PROGRAM Rotina021_Manual
VAR
	status: INT;
	
	posicaoAtual: STRING;
	envialog: STRING;
	
	fbTimeVentila: ton;
	fbTimeAqueci: ton;
	
	totalManual: STRING(255);
	tempo: STRING(255);
	
	Estufa: INT;
	
END_VAR

fbTimeVentila();
fbTimeAqueci();
Estufa:= 2;

CASE status OF

0:
IF gvl_p.arrStatusEstufas[Estufa].startManual AND STRING_TO_DT(gvl.progInicio[Estufa]) <= systemtime_to_dt(gvl.fbGetLocalSystemTime.systemTime)  THEN
	status:= 5;
	
	gvl.bstartchart021:= TRUE;
	gvl_p.zona1setpt_021:= gvl_p.arr_CustomTime_021[0,1];
	gvl_p.zona2setpt_021:= gvl_p.arr_CustomTime_021[0,1];
	gvl.liga_ventilacao_021:= TRUE;
	fbTimeVentila(in:= TRUE, pt:=T#1S);
	
///// GERADOR DE LOG -------------------------------------------------------------

envialog:= 'Programação Manual Iniciada ESTUFA 021';
gvl.logRegister21:= envialog;
	
	gvl_p.etapa_process[Estufa] := 'Inicializando';
	
ELSE
	status:= 0;
	IF gvl_p.arrStatusEstufas[Estufa].start THEN
		gvl_p.etapa_process[Estufa] := gvl.progInicio[Estufa];
	END_IF
END_IF
5:
IF fbTimeVentila.Q THEN
	status:= 10;
	gvl.liga_ventilacao_021:=FALSE;
	fbTimeVentila(in:= FALSE);
ELSE
	status:= 5;
END_IF

10:
IF gvl.ventilacao_Ligada_021 THEN
	status:= 15;
	
	gvl.liga_aquecimento_021:= TRUE;
	fbTimeAqueci(in:= TRUE, pt:= T#1S);
	
///// GERADOR DE LOG -------------------------------------------------------------

envialog:= 'Aquecendo ESTUFA 021';
gvl.logRegister21:= envialog;

	gvl_p.etapa_process[Estufa] := 'Aquecendo';
	
ELSE
	status:= 10;
END_IF

15:
IF fbTimeAqueci.Q THEN
	status:= 20;
	
	gvl.liga_aquecimento_021:= FALSE;
	fbTimeAqueci(in:=false);
ELSE
	status:= 15;
END_IF

20:
IF gvl.zona1atual_021 >= gvl_p.zona1setpt_021 THEN
	status:= 30;
	
gvl.progInicio[Estufa]:= DT_TO_STRING(gvl.somaTempo);
	
///// CALCULAR FIM DA SECAGEM E DA ARMAZENAGEM --------------------------------------------------------------------------------

totalManual:= insert('T#h',INT_TO_STRING(gvl.totalManual[Estufa]),2);
gvl_p.arrStatusEstufas[Estufa].inicioSecagem := STRING_TO_DT(gvl.progInicio[Estufa]);
gvl_p.arrStatusEstufas[Estufa].fimSecagem := STRING_TO_DT(gvl.progInicio[Estufa]) + STRING_TO_TIME(totalManual);
gvl_P.arrStatusEstufas[Estufa].prevFimSeca := gvl_p.arrStatusEstufas[Estufa].fimSecagem;
//gvl_p.arrStatusEstufas[0].fimArmazenagem := gvl_p.arrStatusEstufas[0].fimSecagem + gvl_p.arrStatusEstufas[0].tempoArmazenagem ;

///// IMPRIMIR A HORA E A DATA DO INICIO DA SECAGEM ---------------------------------------------------------------------------
gvl_p.arrStatusEstufas[Estufa].statusInicioSecagem := '';
gvl_p.arrStatusEstufas[Estufa].statusInicioSecagem := concat(gvl_p.arrStatusEstufas[Estufa].statusInicioSecagem,gvl.hora);
gvl_p.arrStatusEstufas[Estufa].statusInicioSecagem := concat(gvl_p.arrStatusEstufas[Estufa].statusInicioSecagem,':');
gvl_p.arrStatusEstufas[Estufa].statusInicioSecagem := concat(gvl_p.arrStatusEstufas[Estufa].statusInicioSecagem,gvl.minuto);
gvl_p.arrStatusEstufas[Estufa].statusInicioSecagem := concat(gvl_p.arrStatusEstufas[Estufa].statusInicioSecagem,' ');
gvl_p.arrStatusEstufas[Estufa].statusInicioSecagem := concat(gvl_p.arrStatusEstufas[Estufa].statusInicioSecagem,gvl.dia);
gvl_p.arrStatusEstufas[Estufa].statusInicioSecagem := concat(gvl_p.arrStatusEstufas[Estufa].statusInicioSecagem,'/');
gvl_p.arrStatusEstufas[Estufa].statusInicioSecagem := concat(gvl_p.arrStatusEstufas[Estufa].statusInicioSecagem,gvl.mes);
gvl_p.arrStatusEstufas[Estufa].statusInicioSecagem := concat(gvl_p.arrStatusEstufas[Estufa].statusInicioSecagem,'/');
gvl_p.arrStatusEstufas[Estufa].statusInicioSecagem := concat(gvl_p.arrStatusEstufas[Estufa].statusInicioSecagem,gvl.ano);

//--------------------REATOR------------------------------------

IF gravarConfigPosicao_Reator.bGravarConfigPosicao_Reator THEN
	gvl_p.arrStatusEstufas[Estufa].inicioReator := '';
	gvl_p.arrStatusEstufas[Estufa].inicioReator := concat(gvl_p.arrStatusEstufas[Estufa].inicioReator,gvl.hora);
	gvl_p.arrStatusEstufas[Estufa].inicioReator := concat(gvl_p.arrStatusEstufas[Estufa].inicioReator,':');
	gvl_p.arrStatusEstufas[Estufa].inicioReator := concat(gvl_p.arrStatusEstufas[Estufa].inicioReator,gvl.minuto);
	gvl_p.arrStatusEstufas[Estufa].inicioReator := concat(gvl_p.arrStatusEstufas[Estufa].inicioReator,' ');
	gvl_p.arrStatusEstufas[Estufa].inicioReator := concat(gvl_p.arrStatusEstufas[Estufa].inicioReator,gvl.dia);
	gvl_p.arrStatusEstufas[Estufa].inicioReator := concat(gvl_p.arrStatusEstufas[Estufa].inicioReator,'/');
	gvl_p.arrStatusEstufas[Estufa].inicioReator := concat(gvl_p.arrStatusEstufas[Estufa].inicioReator,gvl.mes);
	gvl_p.arrStatusEstufas[Estufa].inicioReator := concat(gvl_p.arrStatusEstufas[Estufa].inicioReator,'/');
	gvl_P.arrStatusEstufas[Estufa].inicioReator := concat(gvl_p.arrStatusEstufas[Estufa].inicioReator,gvl.ano);
END_IF

///// DECOMPOR A VARIAVEL FIM DA SECAGEM -----------------------------------------------------------------------------------------------
gvl_p.arrStatusEstufas[Estufa].diaSec := MID(STR:= DT_TO_STRING(gvl_p.arrStatusEstufas[Estufa].fimSecagem) , LEN:= 2, POS:=12);
gvl_p.arrStatusEstufas[Estufa].mesSec := MID(STR:= DT_TO_STRING(gvl_p.arrStatusEstufas[Estufa].fimSecagem), LEN:= 2, POS:=9);
gvl_p.arrStatusEstufas[Estufa].anoSec := MID(STR:= DT_TO_STRING(gvl_p.arrStatusEstufas[Estufa].fimSecagem), LEN:= 2, POS:=6);
gvl_p.arrStatusEstufas[Estufa].horaSec := MID(STR:= DT_TO_STRING(gvl_p.arrStatusEstufas[Estufa].fimSecagem), LEN:= 2, POS:=15);
gvl_p.arrStatusEstufas[Estufa].minutoSec := MID(STR:= DT_TO_STRING(gvl_p.arrStatusEstufas[Estufa].fimSecagem), LEN:= 2, POS:=18);

///// IMPRIMIR A HORA E A DATA DO FIM DA SECAGEM --------------------------------------------------------------------------------------------------------
gvl_p.arrStatusEstufas[Estufa].statusFimSecagem := '';
gvl_p.arrStatusEstufas[Estufa].statusFimSecagem := concat(gvl_p.arrStatusEstufas[Estufa].statusFimSecagem,gvl_p.arrStatusEstufas[0].horaSec);
gvl_p.arrStatusEstufas[Estufa].statusFimSecagem := concat(gvl_p.arrStatusEstufas[Estufa].statusFimSecagem,':');
gvl_p.arrStatusEstufas[Estufa].statusFimSecagem := concat(gvl_p.arrStatusEstufas[Estufa].statusFimSecagem,gvl_p.arrStatusEstufas[0].minutoSec);
gvl_p.arrStatusEstufas[Estufa].statusFimSecagem := concat(gvl_p.arrStatusEstufas[Estufa].statusFimSecagem,' ');
gvl_p.arrStatusEstufas[Estufa].statusFimSecagem := concat(gvl_p.arrStatusEstufas[Estufa].statusFimSecagem,gvl_p.arrStatusEstufas[0].diaSec);
gvl_p.arrStatusEstufas[Estufa].statusFimSecagem := concat(gvl_p.arrStatusEstufas[Estufa].statusFimSecagem,'/');
gvl_p.arrStatusEstufas[Estufa].statusFimSecagem := concat(gvl_p.arrStatusEstufas[Estufa].statusFimSecagem,gvl_p.arrStatusEstufas[0].mesSec);
gvl_p.arrStatusEstufas[Estufa].statusFimSecagem := concat(gvl_p.arrStatusEstufas[Estufa].statusFimSecagem,'/');
gvl_p.arrStatusEstufas[Estufa].statusFimSecagem := concat(gvl_p.arrStatusEstufas[Estufa].statusFimSecagem,gvl_p.arrStatusEstufas[0].anoSec);


///// GERADOR DE LOG -------------------------------------------------------------
envialog:= 'Inicio T1 ESTUFA 021';
gvl.logRegister21:= envialog;

gvl_p.etapa_process[2]:= 'T1';

ELSE
	IF gvl_p.arr_CustomTime_021[1,1] = 0 THEN
		status:= 45;
	END_IF
	status:= 20;
END_IF

30:
tempo:= insert('T#h',INT_TO_STRING(gvl_p.arr_CustomTime_021[1,1]),2);
IF STRING_TO_DT(gvl.progInicio[Estufa]) + STRING_TO_TIME(tempo) = systemtime_to_dt(gvl.fbGetLocalSystemTime.systemTime) THEN
	status:= 31;
	
	gvl_p.zona1setpt_021:= gvl_p.arr_CustomTime_021[0,2];
	gvl_p.zona2setpt_021:= gvl_p.arr_CustomTime_021[0,2];
	gvl.progInicio[Estufa]:= DT_TO_STRING(STRING_TO_DT(gvl.progInicio[Estufa]) + STRING_TO_TIME(tempo));
	
///// GERADOR DE LOG -------------------------------------------------------------
envialog:= 'Inicio T2 ESTUFA 021';
gvl.logRegister21:= envialog;

gvl_p.etapa_process[2]:= 'T2';
	
ELSE
	status:= 30;
END_IF

31:
tempo:= insert('T#h',INT_TO_STRING(gvl_p.arr_CustomTime_021[1,2]),2);
IF STRING_TO_DT(gvl.progInicio[Estufa]) + STRING_TO_TIME(tempo) = systemtime_to_dt(gvl.fbGetLocalSystemTime.systemTime) THEN
	status:= 32;
	
	gvl_p.zona1setpt_021:= gvl_p.arr_CustomTime_021[0,3];
	gvl_p.zona2setpt_021:= gvl_p.arr_CustomTime_021[0,3];
	gvl.progInicio[Estufa]:= DT_TO_STRING(STRING_TO_DT(gvl.progInicio[Estufa]) + STRING_TO_TIME(tempo));
	
///// GERADOR DE LOG -------------------------------------------------------------
envialog:= 'Inicio T3 ESTUFA 021';
gvl.logRegister21:= envialog;

gvl_p.etapa_process[2]:= 'T3';
	
ELSE
	IF gvl_p.arr_CustomTime_021[1,2] = 0 THEN
		status:= 45;
	END_IF
	status:= 31;
END_IF

32:
tempo:= insert('T#h',INT_TO_STRING(gvl_p.arr_CustomTime_021[1,3]),2);
IF STRING_TO_DT(gvl.progInicio[Estufa]) + STRING_TO_TIME(tempo) = systemtime_to_dt(gvl.fbGetLocalSystemTime.systemTime) THEN
	status:= 33;
	
	gvl_p.zona1setpt_021:= gvl_p.arr_CustomTime_021[0,4];
	gvl_p.zona2setpt_021:= gvl_p.arr_CustomTime_021[0,4];
	gvl.progInicio[Estufa]:= DT_TO_STRING(STRING_TO_DT(gvl.progInicio[Estufa]) + STRING_TO_TIME(tempo));
	
///// GERADOR DE LOG -------------------------------------------------------------
envialog:= 'Inicio T4 ESTUFA 021';
gvl.logRegister21:= envialog;

gvl_p.etapa_process[2]:= 'T4';
	
ELSE
	IF gvl_p.arr_CustomTime_021[1,3] = 0 THEN
		status:= 45;
	END_IF
	status:= 32;
END_IF

33:
tempo:= insert('T#h',INT_TO_STRING(gvl_p.arr_CustomTime_021[1,4]),2);
IF STRING_TO_DT(gvl.progInicio[Estufa]) + STRING_TO_TIME(tempo) = systemtime_to_dt(gvl.fbGetLocalSystemTime.systemTime) THEN
	status:= 34;
	
	gvl_p.zona1setpt_021:= gvl_p.arr_CustomTime_021[0,5];
	gvl_p.zona2setpt_021:= gvl_p.arr_CustomTime_021[0,5];
	gvl.progInicio[Estufa]:= DT_TO_STRING(STRING_TO_DT(gvl.progInicio[Estufa]) + STRING_TO_TIME(tempo));
	
///// GERADOR DE LOG -------------------------------------------------------------
envialog:= 'Inicio T5 ESTUFA 021';
gvl.logRegister21:= envialog;

gvl_p.etapa_process[2]:= 'T5';
	
ELSE
	IF gvl_p.arr_CustomTime_021[1,4] = 0 THEN
		status:= 45;
	END_IF
	status:= 33;
END_IF

34:
tempo:= insert('T#h',INT_TO_STRING(gvl_p.arr_CustomTime_021[1,5]),2);
IF STRING_TO_DT(gvl.progInicio[Estufa]) + STRING_TO_TIME(tempo) = systemtime_to_dt(gvl.fbGetLocalSystemTime.systemTime) THEN
	status:= 35;
	
	gvl_p.zona1setpt_021:= gvl_p.arr_CustomTime_021[0,6];
	gvl_p.zona2setpt_021:= gvl_p.arr_CustomTime_021[0,6];
	gvl.progInicio[Estufa]:= DT_TO_STRING(STRING_TO_DT(gvl.progInicio[Estufa]) + STRING_TO_TIME(tempo));
	
///// GERADOR DE LOG -------------------------------------------------------------
envialog:= 'Inicio T6 ESTUFA 021';
gvl.logRegister21:= envialog;

gvl_p.etapa_process[2]:= 'T6';
	
ELSE
	IF gvl_p.arr_CustomTime_021[1,5] = 0 THEN
		status:= 45;
	END_IF
	status:= 34;
END_IF

35:
tempo:= insert('T#h',INT_TO_STRING(gvl_p.arr_CustomTime_021[1,6]),2);
IF STRING_TO_DT(gvl.progInicio[Estufa]) + STRING_TO_TIME(tempo) = systemtime_to_dt(gvl.fbGetLocalSystemTime.systemTime) THEN
	status:= 36;
	
	gvl_p.zona1setpt_021:= gvl_p.arr_CustomTime_021[0,7];
	gvl_p.zona2setpt_021:= gvl_p.arr_CustomTime_021[0,7];
	gvl.progInicio[Estufa]:= DT_TO_STRING(STRING_TO_DT(gvl.progInicio[Estufa]) + STRING_TO_TIME(tempo));
	
///// GERADOR DE LOG -------------------------------------------------------------
envialog:= 'Inicio T7 ESTUFA 021';
gvl.logRegister21:= envialog;

gvl_p.etapa_process[2]:= 'T7';
	
ELSE
	IF gvl_p.arr_CustomTime_021[1,6] = 0 THEN
		status:= 45;
	END_IF
	status:= 35;
END_IF

36:
tempo:= insert('T#h',INT_TO_STRING(gvl_p.arr_CustomTime_021[1,7]),2);
IF STRING_TO_DT(gvl.progInicio[Estufa]) + STRING_TO_TIME(tempo) = systemtime_to_dt(gvl.fbGetLocalSystemTime.systemTime) THEN
	status:= 37;
	
	gvl_p.zona1setpt_021:= gvl_p.arr_CustomTime_021[0,8];
	gvl_p.zona2setpt_021:= gvl_p.arr_CustomTime_021[0,8];
	gvl.progInicio[Estufa]:= DT_TO_STRING(STRING_TO_DT(gvl.progInicio[Estufa]) + STRING_TO_TIME(tempo));
	
///// GERADOR DE LOG -------------------------------------------------------------
envialog:= 'Inicio T8 ESTUFA 021';
gvl.logRegister21:= envialog;

gvl_p.etapa_process[2]:= 'T8';
	
ELSE
	IF gvl_p.arr_CustomTime_021[1,7] = 0 THEN
		status:= 45;
	END_IF
	status:= 36;
END_IF

37:
tempo:= insert('T#h',INT_TO_STRING(gvl_p.arr_CustomTime_021[1,8]),2);
IF STRING_TO_DT(gvl.progInicio[Estufa]) + STRING_TO_TIME(tempo) = systemtime_to_dt(gvl.fbGetLocalSystemTime.systemTime) THEN
	status:= 38;
	
	gvl_p.zona1setpt_021:= gvl_p.arr_CustomTime_021[0,9];
	gvl_p.zona2setpt_021:= gvl_p.arr_CustomTime_021[0,9];
	gvl.progInicio[Estufa]:= DT_TO_STRING(STRING_TO_DT(gvl.progInicio[Estufa]) + STRING_TO_TIME(tempo));
	
///// GERADOR DE LOG -------------------------------------------------------------
envialog:= 'Inicio T9 ESTUFA 021';
gvl.logRegister21:= envialog;

gvl_p.etapa_process[2]:= 'T9';
	
ELSE
	IF gvl_p.arr_CustomTime_021[1,8] = 0 THEN
		status:= 45;
	END_IF
	status:= 37;
END_IF

38:
tempo:= insert('T#h',INT_TO_STRING(gvl_p.arr_CustomTime_021[1,9]),2);
IF STRING_TO_DT(gvl.progInicio[Estufa]) + STRING_TO_TIME(tempo) = systemtime_to_dt(gvl.fbGetLocalSystemTime.systemTime) THEN
	status:= 40;
	
	gvl_p.zona1setpt_021:= gvl_p.arr_CustomTime_021[0,10];
	gvl_p.zona2setpt_021:= gvl_p.arr_CustomTime_021[0,10];
	gvl.progInicio[Estufa]:= DT_TO_STRING(STRING_TO_DT(gvl.progInicio[Estufa]) + STRING_TO_TIME(tempo));
	
///// GERADOR DE LOG -------------------------------------------------------------
envialog:= 'Inicio T10 ESTUFA 021';
gvl.logRegister21:= envialog;

gvl_p.etapa_process[2]:= 'T10';
	
ELSE
	IF gvl_p.arr_CustomTime_021[1,9] = 0 THEN
		status:= 45;
	END_IF
	status:= 38;
END_IF

40:
tempo:= insert('T#h',INT_TO_STRING(gvl_p.arr_CustomTime_021[1,10]),2);
IF STRING_TO_DT(gvl.progInicio[Estufa]) + STRING_TO_TIME(tempo) = systemtime_to_dt(gvl.fbGetLocalSystemTime.systemTime) THEN
	status:= 50;
	
	gvl_p.arrStatusEstufas[Estufa].startManual:= FALSE;
	gvl.bstartchart021:= FALSE;
	gvl.desl_aquecimento_021:= TRUE;
	fbTimeAqueci(in:=TRUE, pt:=T#1S);
	
	gvl_p.etapa_process[Estufa] := '';
	
	gvl_p.arrStatusEstufas[Estufa].statusInicioSecagem := '';
	gvl_p.arrStatusEstufas[Estufa].inicioReator := '';
	gvl_p.arrStatusEstufas[Estufa].statusFimSecagem := '';
	gvl_p.arrStatusEstufas[Estufa].statusFimArmazenagem := '';
	gvl_p.arrStatusEstufas[Estufa].fimSecagem:= DT#1970-1-1-0:0:0;
	gvl.endArm21:= T#0S;
	gvl.endSeca21:= T#0S;
	
///// GERADOR DE LOG -------------------------------------------------------------
envialog:= 'Programação Finalizada ESTUFA 021';
gvl.logRegister21:= envialog;

gvl_p.etapa_process[2]:= '';

ELSE
	IF gvl_p.arr_CustomTime_021[1,10] = 0 THEN
		status:= 45;
	END_IF
	status:= 40;
END_IF

45:
IF gvl_p.arrStatusEstufas[Estufa].startManual THEN
status:= 50;
	
	gvl_p.arrStatusEstufas[Estufa].startManual:= FALSE;
	gvl.bstartchart021:= FALSE;
	gvl.desl_aquecimento_021:= TRUE;
	fbTimeAqueci(in:=TRUE, pt:=T#1S);
	
	gvl_p.etapa_process[Estufa] := '';
	
	gvl_p.arrStatusEstufas[Estufa].statusInicioSecagem := '';
	gvl_p.arrStatusEstufas[Estufa].inicioReator := '';
	gvl_p.arrStatusEstufas[Estufa].statusFimSecagem := '';
	gvl_p.arrStatusEstufas[Estufa].statusFimArmazenagem := '';
	gvl_p.arrStatusEstufas[Estufa].fimSecagem:= DT#1970-1-1-0:0:0;
	gvl.endArm21:= T#0S;
	gvl.endSeca21:= T#0S;
	
///// GERADOR DE LOG -------------------------------------------------------------
envialog:= 'Programação Finalizada ESTUFA 021';
gvl.logRegister21:= envialog;

gvl_p.etapa_process[2]:= '';

ELSE
	status:= 45;
END_IF

50:
IF fbTimeAqueci.Q THEN
	status:= 0;
	
	gvl.desl_aquecimento_021:= FALSE;
	fbTimeAqueci(in:= FALSE);
	
ELSE
	status:= 50;
END_IF
END_CASE

END_PROGRAM

(* stored: Version 1.1.0.1, ProductVersion 3.1.4024.12
   POU Rotina021_Manual: Id {bd52bb73-9ca1-4598-a17c-97bc04f5778f}, SpecialFunc None *)
